Fanuc KAREL source: kt00177.KL

-- PROVISIONAL review KL for V940-1; original PC SHA256 b64ea2c52aeabb51c7ec7e28431f201506f64052cf6f67b73cf8dcffd8cee47e
-- Incomplete behavior may be omitted. Consult companion uncertainty JSON. Do not deploy.
PROGRAM KT00177
%NOLOCKGROUP
VAR
  I2 : INTEGER
  OUT : INTEGER
-- UNRESOLVED_DECL Y1 type=002018
BEGIN
  -- V9_ZERO_TABLE_METADATA_HINT layout=0001; no indexed target words; source/name/runtime held
  -- UNRESOLVED_PC offsets 5-19; opcodes 2E,22,9D,33,B2
  -- UNRESOLVED_PC offsets 24-35; opcodes 2E,23
  -- UNRESOLVED_PC offsets 40-62; opcodes 22,9D,33,B1,21,56,23
  -- UNRESOLVED_PC offsets 67-71; opcodes 7F
END KT00177
